FUNCTION_BLOCK FB_Multiply2Ints
VAR_INPUT
	Int1	: INT;
	Int2	: INT;
END_VAR
VAR_OUTPUT
	Result	: INT;
END_VAR

Result := Int1 * Int2;

END_FUNCTION_BLOCK

(* stored: Version 1.1.0.1, ProductVersion 3.1.4024.12
   POU FB_Multiply2Ints: Id {39965b16-741e-4a23-bd9e-5ff20d8c9780}, SpecialFunc None *)
